FUNCTION F_FormatString : String
VAR_INPUT
	sInput,
	sPrefix		:STRING;
	nLenght		:INT;
END_VAR
VAR
	nPosition	:INT;
END_VAR

nPosition := FIND(sInput,sPrefix);
F_FormatString := LEFT(sInput,(nPosition + nLenght));

END_FUNCTION

(* stored: Version 1.1.0.1, ProductVersion 3.1.4024.11
   POU F_FormatString: Id {094edad2-808e-4b5e-9920-ea4de8c02573}, SpecialFunc None *)
